// TIA Portal project "HorasyFechas" (V16)

(* hardware
DEVICE "S7-1200 station_1"  S7-1200 Station
   slot 0: "Rack_0"  S7-1200 Rack  Rack  V1.0
   slot 1: "PLC_1"  CPU 1214C AC/DC/Rly  6ES7 214-1BG40-0XB0  V4.4
*)

// ===== PLC "PLC_1"  CPU 1214C AC/DC/Rly =====

VAR_GLOBAL   // PLC tag table "Tabla de variables estándar"
   "Tag_1" AT %I0.0 : Bool;
   "Tag_2" AT %MW100 : Int;
   "Tag_3" AT %I0.1 : Bool;
   "Tag_4" AT %MW104 : Int;
   "Tag_5" AT %M0.0 : Bool;
   "Tag_6" AT %MW108 : Int;
   "Tag_7" AT %MW112 : Int;
   "Tag_8" AT %Q0.0 : Bool;
END_VAR

DATA_BLOCK "FECHA Y HORA"   // DB1
{ S7_Optimized_Access := 'TRUE' }
VERSION : 0.1
   VAR
      SISTEMA : DTL;
      LOCAL : DTL;
   END_VAR
BEGIN
END_DATA_BLOCK

ORGANIZATION_BLOCK "Main"   // OB1, LAD, ProgramCycle
TITLE = "Main Program Sweep (Cycle)"
{ S7_Optimized_Access := 'TRUE' }
VERSION : 0.1
   VAR_INPUT
      Initial_Call : Bool;   // Initial call of this OB
      Remanence : Bool;   // =True, if remanent data are available
   END_VAR
BEGIN

REGION Network 1
   // Escribir o modificar la hora y fecha del sistema o local
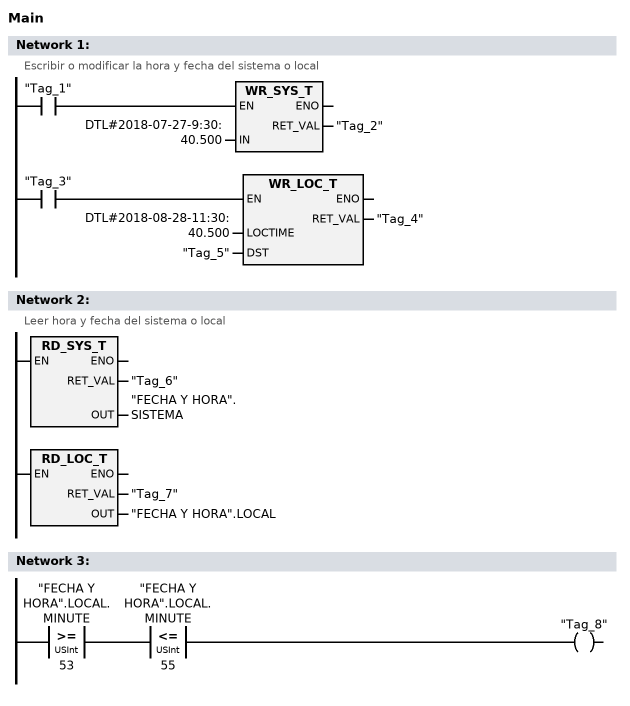
   IF "Tag_1" THEN "Tag_2" := WR_SYS_T(IN := DTL#2018-07-27-9:30:40.500); END_IF;
   IF "Tag_3" THEN "Tag_4" := WR_LOC_T(LOCTIME := DTL#2018-08-28-11:30:40.500, DST := "Tag_5"); END_IF;
END_REGION

REGION Network 2
   // Leer hora y fecha del sistema o local
   "Tag_6" := RD_SYS_T(OUT => "FECHA Y HORA".SISTEMA);
   "Tag_7" := RD_LOC_T(OUT => "FECHA Y HORA".LOCAL);
END_REGION

REGION Network 3
   RUNG wire#powerrail
      { S7_Templates := "SrcType := USInt" } GE_Contact(in1 := "FECHA Y HORA".LOCAL.MINUTE, in2 := 53)
      { S7_Templates := "SrcType := USInt" } LE_Contact(in1 := "FECHA Y HORA".LOCAL.MINUTE, in2 := 55)
      Coil( "Tag_8" )
   END_RUNG
   // the same network as SCL:
   "Tag_8" := ("FECHA Y HORA".LOCAL.MINUTE >= 53) AND ("FECHA Y HORA".LOCAL.MINUTE <= 55);
END_REGION
END_ORGANIZATION_BLOCK